{attribute 'qualified_only'}
{attribute 'strict'}
TYPE
    eTcoLoggerTests :
    (
		Push := 10,
		PushMultiple := 20,
		PushMultipleInMoreCycles := 30
    );
END_TYPE

(* stored: Version 1.1.0.1, ProductVersion 3.1.4024.9
   DUT eTcoLoggerTests: Id {3152a930-9ddc-047f-03f1-d36a10a1ade6} *)
